PROGRAM MAIN
VAR
fbEditLineInFile : FB_EditLineInFile;
   
    sFilePath    : STRING := 'C:\recipe\Receita01.txt';
    sNewText     : STRING(255) := 'LINHA 50 ATUALIZADA$R$N';
	bStart: BOOL;
	nErrorId: UDINT;
	bError: BOOL;
END_VAR

fbEditLineInFile(
	sFilePath:= sFilePath, 
	nLineToEdit:= 10, 
	sNewContent:= sNewText, 
	bStart:= bStart, 
	bDone=> , 
	bBusy=> , 
	bError=> bError, 
	nErrorId=> nErrorId);

END_PROGRAM

(* stored: Version 1.1.0.1
   POU MAIN: Id {8e9ff765-9723-4021-8d6a-9e1f73b0e85c}, SpecialFunc None *)
